FUNCTION_BLOCK Test_AssertEquals_PVOID EXTENDS T_UnitTestBase
VAR
    AssertionUnderTest : T_Assertion;
    PVOID_Variable : PVOID := 1111;
END_VAR

// Test the assertion...
AssertionUnderTest.AssertEquals_PVOID(
    Expected := 2222,
    Actual   := PVOID_Variable,
    VariableName := 'PVOID_Variable'); 
    
// Assert that the assertion failed...
Assertion.AssertEquals_BOOL(Expected     := TRUE,
                            Actual       := AssertionUnderTest.AssertionFailed,
                            VariableName := 'AssertionUnderTest.AssertionFailed');

// Check the assertion worked...  
CheckAssertion(NextState := 0);

END_FUNCTION_BLOCK

(* stored: Version 1.1.0.1, ProductVersion 3.1.4024.11
   POU Test_AssertEquals_PVOID: Id {7a491631-649a-4653-90e0-541a7c2b8cd4}, SpecialFunc None *)
